// SIMATIC S7-200 project (STEP 7-Micro/WIN), CPU 221 REL 01.10

ORGANIZATION_BLOCK 主程序:OB1
TITLE=程序注释
BEGIN
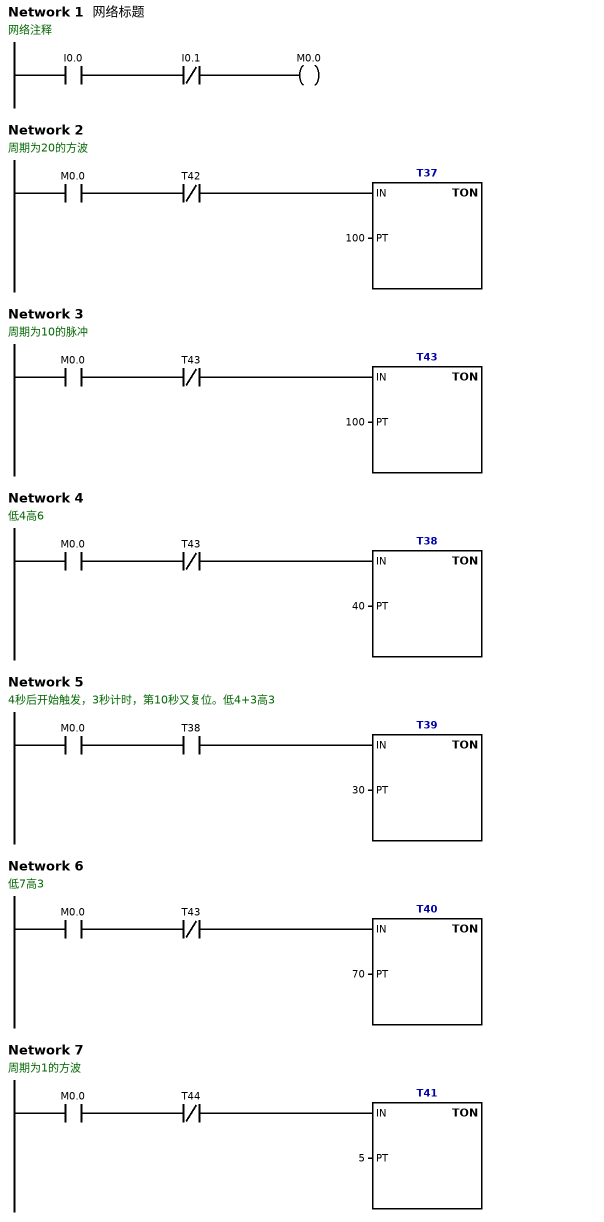
Network 1 // 网络标题
// 网络注释
LD     I0.0
AN     I0.1
=      M0.0
Network 2
// 周期为20的方波 
LD     M0.0
AN     T42
TON    T37, 100
Network 3
// 周期为10的脉冲
LD     M0.0
AN     T43
TON    T43, 100
Network 4
// 低4高6
LD     M0.0
AN     T43
TON    T38, 40
Network 5
// 4秒后开始触发，3秒计时，第10秒又复位。低4+3高3
LD     M0.0
A      T38
TON    T39, 30
Network 6
// 低7高3
LD     M0.0
AN     T43
TON    T40, 70
Network 7
// 周期为1的方波
LD     M0.0
AN     T44
TON    T41, 5
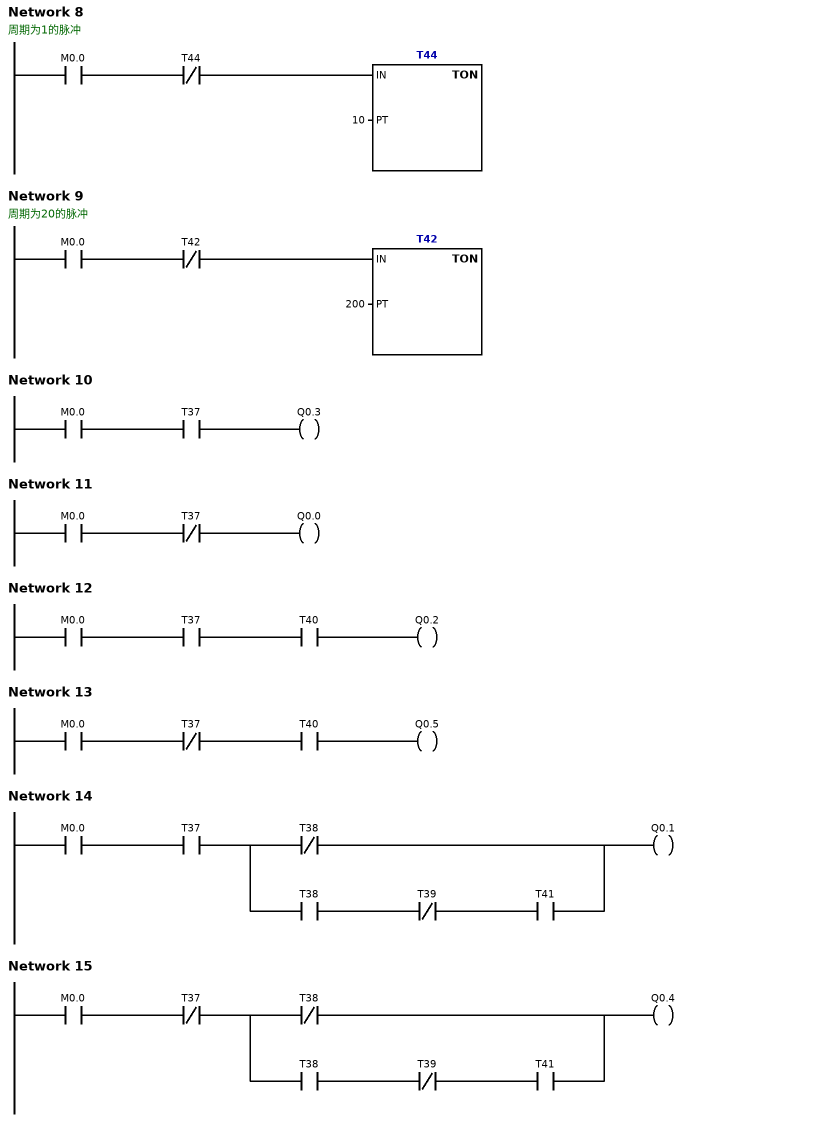
Network 8
// 周期为1的脉冲
LD     M0.0
AN     T44
TON    T44, 10
Network 9
// 周期为20的脉冲
LD     M0.0
AN     T42
TON    T42, 200
Network 10
LD     M0.0
A      T37
=      Q0.3
Network 11
LD     M0.0
AN     T37
=      Q0.0
Network 12
LD     M0.0
A      T37
A      T40
=      Q0.2
Network 13
LD     M0.0
AN     T37
A      T40
=      Q0.5
Network 14
LD     M0.0
A      T37
LDN    T38
LD     T38
AN     T39
A      T41
OLD
ALD
=      Q0.1
Network 15
LD     M0.0
AN     T37
LDN    T38
LD     T38
AN     T39
A      T41
OLD
ALD
=      Q0.4
END_ORGANIZATION_BLOCK
